INTERFACE IStation

METHOD HasMover : BOOL
VAR_INPUT
END_VAR
END_METHOD

METHOD IsClear : BOOL
VAR_INPUT
END_VAR
END_METHOD

METHOD isComplete : BOOL
VAR_INPUT
END_VAR
END_METHOD

METHOD IsOperating : BOOL
VAR_INPUT
END_VAR
END_METHOD

METHOD IsReady : BOOL
VAR_INPUT
END_VAR
END_METHOD

PROPERTY Position : MC_LREAL
GET
END_GET
SET
END_SET
END_PROPERTY

END_INTERFACE

(* stored: Version 1.1.0.1, ProductVersion 3.1.4024.9
   Itf IStation: Id {d53abde8-a061-4411-9fc7-d7a9304584ff}
   Method HasMover: Id {bbc535d0-db75-4784-af7a-7fdceacdeede}
   Method IsClear: Id {3bd7b012-e144-45f5-baa9-13115e740b45}
   Method isComplete: Id {5ff9ac5b-9b0a-4f0e-9ce4-355e0f44f07f}
   Method IsOperating: Id {022d1ae7-70eb-4d51-934d-8d448efa527f}
   Method IsReady: Id {4d8fc97e-69c4-498f-a021-ba3fb6f5743f}
   Property Position: Id {3e9be7e9-e67d-46c2-81c2-a99de33f0222}
   Get Get: Id {99828a85-cb6c-467b-9b04-6d446a05124f}
   Set Set: Id {4228f819-bdd1-41e4-aa7f-1b2439f45f7b} *)
